TYPE ST_HW_InputsSubsystemManager :
(**************************************************************************************
 * 	Application		:	Framework
 *	Revision		:	$Revision: 404529 $
 *	Revision date	:	$Date: 2018-04-23 08:21:38 +0200 (Mo., 23 Apr 2018) $
 *	Last changed by	:	$Author: b7bolm $
 *	URL				:	$URL: http://almscdc.swisslog.com/repo/SWPD/Development/BoxControlFramework/20_Release/trunk/01_Software/BCF/BCF/JumpStart/20_Product/10_App/15_Subsystem/10_Lib/10_Conv/01_DUTs/10_Dummy/ST_HW_InputsSubSystemManager.TcDUT $
 *
 *	Purpose			:	Subsystem Manager - Hardware inputs
 *
 * ------------------------------------------------------------------------------------
 *	Copyright Swisslog [IP AG], Switzerland. All rights reserved.
 * 
 * ------------------------------------------------------------------------------------
 *	
 * 	Revision History: 
 *
 * 	VERSION			DATE			INITIALS			DESCRIPTION
 *	0.1				01.01.2001		swl					Example
 *
 **************************************************************************************)
STRUCT
	EtherCAT_MasterState			AT %I* : UINT; // Diagnostic info of EtherCat Master node 
	EtherCAT_MasterWorkingCounter	AT %I* : UINT; // Diagnostic info of EtherCat Master node 
	DeviceState	  					AT %I* : ARRAY [1..400] OF UINT; // Diagnostic info of EtherCAT slave devices
END_STRUCT
END_TYPE

(* stored: Version 1.1.0.1, ProductVersion 3.1.4022.12
   DUT ST_HW_InputsSubSystemManager: Id {60125919-c6f2-4048-b3fc-9ebfe3d58f67} *)
